FUNCTION_BLOCK TEST_ADD (* Test ADD functions *)
  (* Standard: IEC 61499-1 *)
  (* Version 0.0, 2006-09-11, JHC, Holobloc Inc *)
  (* Compiler header: package fb.rt.test; *)
  (* Compiler classdef: SimpleFB *)
  (* Compiler Java Sun JDK 1.5.0 *)
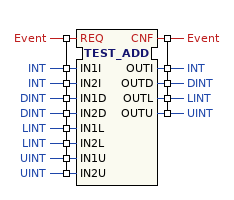
  EVENT_INPUT
    REQ WITH IN1I, IN2I, IN2D, IN1L, IN2L, IN1U, IN2U, IN1D;
  END_EVENT
  EVENT_OUTPUT
    CNF WITH OUTI, OUTD, OUTL, OUTU;
  END_EVENT
  VAR_INPUT
    IN1I : INT;
    IN2I : INT;
    IN1D : DINT;
    IN2D : DINT;
    IN1L : LINT;
    IN2L : LINT;
    IN1U : UINT;
    IN2U : UINT;
  END_VAR
  VAR_OUTPUT
    OUTI : INT;
    OUTD : DINT;
    OUTL : LINT;
    OUTU : UINT;
  END_VAR
  ALGORITHM REQ IN FBD:
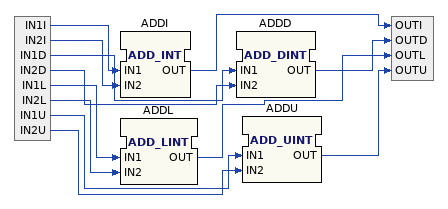
    FBS
      ADDI : ADD_INT;
      ADDD : ADD_DINT;
      ADDL : ADD_LINT;
      ADDU : ADD_UINT;
    END_FBS
    DATA_CONNECTIONS
      IN1I TO ADDI.IN1;
      IN2I TO ADDI.IN2;
      ADDI.OUT TO OUTI;
      IN1D TO ADDD.IN1;
      IN2D TO ADDD.IN2;
      ADDD.OUT TO OUTD;
      IN1L TO ADDL.IN1;
      IN2L TO ADDL.IN2;
      ADDL.OUT TO OUTL;
      IN1U TO ADDU.IN1;
      IN2U TO ADDU.IN2;
      ADDU.OUT TO OUTU;
    END_CONNECTIONS
  END_ALGORITHM
END_FUNCTION_BLOCK
